{attribute 'qualified_only'}
{attribute 'strict'}
{attribute 'to_string'}
TYPE
ApproachScenario_e :
(
    WaitOnFinishedProcess,
    WaitOnFreeStation,
    DoNotWait,
    WaitOnPrevProcess,
    WaitOnExternalTrigger,
    _MAX
);
END_TYPE

(* stored: Version 1.1.0.1, ProductVersion 3.1.4024.6
   EnumerationTextList ApproachScenario_e: Id {74e9dac0-84d0-407a-9cbf-53cc751322c7} *)
